TYPE UDT_AxisAdmin :
STRUCT
	i: UDT_AXISinput;
	o: UDT_AXISOUTPUT;
	Axis: Axis_Ref;
END_STRUCT
END_TYPE

(* stored: Version 1.1.0.1, ProductVersion 3.1.4022.16
   DUT UDT_AxisAdmin: Id {276e6697-6418-414a-8f33-d557a894c691} *)
